FUNCTION_BLOCK FB_VisuSim
VAR_INPUT
	bConveyor : BOOL;
END_VAR
VAR_OUTPUT
	bBottle : BOOL;
END_VAR
VAR
	fPos : REAL;
END_VAR

IF bConveyor THEN
	fPos := fPos + 0.1;
END_IF

IF fPos >= 100.0 THEN
	fPos := 0;
END_IF

bBottle := fPos >= 60.0 AND fPos <= 80.0;

END_FUNCTION_BLOCK

(* stored: Version 1.1.0.1, ProductVersion 3.1.4024.12
   POU FB_VisuSim: Id {3774dbef-c7d2-4a4d-811e-1fba5257b332}, SpecialFunc None *)
